(* IEC 61131-3 sources: RegAx/src, 7 files *)

(* ---- RegexCharClass.st ---- *)
NAMESPACE Simatic.Ax.RegAx

    /// Parsed representation of a character class like [abc], [a-z] or [^abc].
    TYPE INTERNAL RegexCharClass : STRUCT
        isNegated : BOOL;
        literalCount : INT;
        literals : ARRAY[1..16] OF CHAR;
        rangeCount : INT;
        ranges : ARRAY[1..8] OF RegexCharClassRange;
    END_STRUCT;
    END_TYPE

END_NAMESPACE

(* ---- RegexCharClassRange.st ---- *)
NAMESPACE Simatic.Ax.RegAx

    /// Inclusive character range used inside a character class.
    TYPE INTERNAL RegexCharClassRange : STRUCT
        rangeStart : CHAR;
        rangeEnd : CHAR;
    END_STRUCT;
    END_TYPE

END_NAMESPACE

(* ---- RegexToken.st ---- *)
NAMESPACE Simatic.Ax.RegAx

    /// Parsed token with optional quantifier information.
    TYPE PUBLIC RegexToken : STRUCT
        tokenType : RegexTokenType;
        literal : CHAR;
        minCount : INT;
        maxCount : INT;
        charClass : RegexCharClass;
    END_STRUCT;
    END_TYPE

END_NAMESPACE

(* ---- RegexTokenType.st ---- *)
NAMESPACE Simatic.Ax.RegAx

    /// Token kinds used by the internal regex tokenizer.
    TYPE PUBLIC RegexTokenType : (
        None,
        Literal,
        DigitClass,
        WordClass,
        CharacterClass,
        EscapedLiteral,
        AnchorStart,
        AnchorEnd
    );
    END_TYPE

END_NAMESPACE

(* ---- Regex.st ---- *)
USING System.Strings;

NAMESPACE Simatic.Ax.RegAx

    /// Public regex facade for configuring a pattern, assigning input and retrieving the match.
    CLASS PUBLIC Regex
        VAR
            /// Pattern used for the next match operation.
            _pattern : STRING;

            /// Input string used for the next match operation.
            _input : STRING;

            /// Last matched substring.
            _match : STRING;

            /// 1-based start index of the last successful match.
            _matchStartIndex : INT;

            /// 1-based end index of the last successful match.
            _matchEndIndex : INT;

            /// Next input position used by MatchNext.
            _nextSearchStartIndex : INT;

            /// Internal tokenizer instance.
            _tokenizer : RegexTokenizer;

            /// Internal matcher instance.
            _matcher : RegexMatcher;
        END_VAR

        /// Stores the regex pattern for subsequent Match calls.
        METHOD PUBLIC SetPattern
            VAR_INPUT
                /// Regex pattern to evaluate.
                pattern : STRING;
            END_VAR
            _pattern := pattern;
        END_METHOD

        /// Stores the input string for subsequent Match calls.
        METHOD PUBLIC SetInput
            VAR_INPUT
                /// Input string to search in.
                inputStr : STRING;
            END_VAR
            _input := inputStr;
            _match := '';
            _matchStartIndex := 0;
            _matchEndIndex := 0;
            _nextSearchStartIndex := 1;
        END_METHOD

        /// Evaluates the configured pattern against the configured input.
        METHOD PUBLIC Match : BOOL
            VAR
                tokens : ARRAY[1..64] OF RegexToken;
                tokenCount : INT;
                anchorStart : BOOL;
                anchorEnd : BOOL;
                inputLength : INT;
                startIndex : INT;
                endIndex : INT;
            END_VAR

            _match := '';
            _matchStartIndex := 0;
            _matchEndIndex := 0;
            _nextSearchStartIndex := 1;
            IF NOT _tokenizer.Tokenize(pattern := _pattern, tokens => tokens, tokenCount => tokenCount, anchorStart => anchorStart, anchorEnd => anchorEnd) THEN
                Match := FALSE;
                RETURN;
            END_IF;

            inputLength := LengthOf(_input);
            IF tokenCount <= 0 THEN
                Match := FALSE;
                RETURN;
            END_IF;

            IF anchorStart THEN
                startIndex := 1;
                IF _matcher.TryMatchFrom(input := _input, startIndex := startIndex, inputLength := inputLength, tokens := tokens, tokenCount := tokenCount, anchorEnd := anchorEnd, endIndex => endIndex) THEN
                    _match := _matcher.BuildMatch(input := _input, startIndex := startIndex, endIndex := endIndex);
                    _matchStartIndex := startIndex;
                    _matchEndIndex := endIndex;
                    _nextSearchStartIndex := endIndex + 1;
                    Match := TRUE;
                    RETURN;
                END_IF;
                Match := FALSE;
                RETURN;
            END_IF;

            startIndex := 1;
            WHILE startIndex <= inputLength DO
                IF _matcher.TryMatchFrom(input := _input, startIndex := startIndex, inputLength := inputLength, tokens := tokens, tokenCount := tokenCount, anchorEnd := anchorEnd, endIndex => endIndex) THEN
                    _match := _matcher.BuildMatch(input := _input, startIndex := startIndex, endIndex := endIndex);
                    _matchStartIndex := startIndex;
                    _matchEndIndex := endIndex;
                    _nextSearchStartIndex := endIndex + 1;
                    Match := TRUE;
                    RETURN;
                END_IF;
                startIndex := startIndex + 1;
            END_WHILE;

            Match := FALSE;
        END_METHOD

        /// Continues searching after the previous successful match.
        METHOD PUBLIC MatchNext : BOOL
            VAR
                tokens : ARRAY[1..64] OF RegexToken;
                tokenCount : INT;
                anchorStart : BOOL;
                anchorEnd : BOOL;
                inputLength : INT;
                startIndex : INT;
                endIndex : INT;
            END_VAR

            _match := '';
            _matchStartIndex := 0;
            _matchEndIndex := 0;

            IF NOT _tokenizer.Tokenize(pattern := _pattern, tokens => tokens, tokenCount => tokenCount, anchorStart => anchorStart, anchorEnd => anchorEnd) THEN
                MatchNext := FALSE;
                RETURN;
            END_IF;

            IF anchorStart OR anchorEnd THEN
                MatchNext := FALSE;
                RETURN;
            END_IF;

            inputLength := LengthOf(_input);
            startIndex := _nextSearchStartIndex;
            IF startIndex < 1 THEN
                startIndex := 1;
            END_IF;

            WHILE startIndex <= inputLength DO
                IF _matcher.TryMatchFrom(input := _input, startIndex := startIndex, inputLength := inputLength, tokens := tokens, tokenCount := tokenCount, anchorEnd := FALSE, endIndex => endIndex) THEN
                    _match := _matcher.BuildMatch(input := _input, startIndex := startIndex, endIndex := endIndex);
                    _matchStartIndex := startIndex;
                    _matchEndIndex := endIndex;
                    _nextSearchStartIndex := endIndex + 1;
                    MatchNext := TRUE;
                    RETURN;
                END_IF;
                startIndex := startIndex + 1;
            END_WHILE;

            MatchNext := FALSE;
        END_METHOD

        /// Returns the substring captured by the last successful Match call.
        METHOD PUBLIC GetMatch : STRING
            GetMatch := _match;
        END_METHOD

        /// Returns the 1-based start index of the last successful match.
        METHOD PUBLIC GetMatchStartIndex : INT
            GetMatchStartIndex := _matchStartIndex;
        END_METHOD

        /// Returns the 1-based end index of the last successful match.
        METHOD PUBLIC GetMatchEndIndex : INT
            GetMatchEndIndex := _matchEndIndex;
        END_METHOD
    END_CLASS

END_NAMESPACE

(* ---- RegexMatcher.st ---- *)
USING System.Strings;

NAMESPACE Simatic.Ax.RegAx

    {axcode:docs-v0:@simatic-ax/regax:Regex.md}
    /// Internal matcher for the supported iterative regex subset.
    CLASS INTERNAL RegexMatcher
        VAR CONSTANT
            /// Maximum length of a returned match.
            MAX_MATCH_LENGTH : INT := 254;
        END_VAR

        /// Tries to match a tokenized pattern against the input string.
        METHOD PUBLIC MatchTokens : BOOL
            VAR_INPUT
                /// Input string to search in.
                input : STRING;

                /// Tokenized regex pattern.
                tokens : ARRAY[1..64] OF RegexToken;

                /// Number of valid tokens.
                tokenCount : INT;

                /// TRUE when matching must start at the beginning of the input.
                anchorStart : BOOL;

                /// TRUE when matching must end at the end of the input.
                anchorEnd : BOOL;
            END_VAR
            VAR_OUTPUT
                /// Matched substring when a match is found.
                matchedText : STRING;
            END_VAR
            VAR
                inputLength : INT;
                startIndex : INT;
                endIndex : INT;
            END_VAR

            MatchTokens := FALSE;
            matchedText := '';
            inputLength := LengthOf(input);

            IF tokenCount <= 0 THEN
                RETURN;
            END_IF;

            IF anchorStart THEN
                startIndex := 1;
                IF THIS.TryMatchFrom(input := input, startIndex := startIndex, inputLength := inputLength, tokens := tokens, tokenCount := tokenCount, anchorEnd := anchorEnd, endIndex => endIndex) THEN
                    matchedText := THIS.BuildMatch(input := input, startIndex := startIndex, endIndex := endIndex);
                    MatchTokens := TRUE;
                END_IF;
                RETURN;
            END_IF;

            startIndex := 1;
            WHILE startIndex <= inputLength DO
                IF THIS.TryMatchFrom(input := input, startIndex := startIndex, inputLength := inputLength, tokens := tokens, tokenCount := tokenCount, anchorEnd := anchorEnd, endIndex => endIndex) THEN
                    matchedText := THIS.BuildMatch(input := input, startIndex := startIndex, endIndex := endIndex);
                    MatchTokens := TRUE;
                    RETURN;
                END_IF;
                startIndex := startIndex + 1;
            END_WHILE;
        END_METHOD

        /// Attempts a match from a specific input position.
        METHOD INTERNAL TryMatchFrom : BOOL
            VAR_INPUT
                /// Input string to search in.
                input : STRING;

                /// 1-based start position for this attempt.
                startIndex : INT;

                /// Cached input length.
                inputLength : INT;

                /// Tokenized regex pattern.
                tokens : ARRAY[1..64] OF RegexToken;

                /// Number of valid tokens.
                tokenCount : INT;

                /// TRUE when the match must consume the full remaining input.
                anchorEnd : BOOL;
            END_VAR
            VAR_OUTPUT
                /// Inclusive end index of the match.
                endIndex : INT;
            END_VAR
            VAR
                tokenIndex : INT;
                inputIndex : INT;
                repeatCount : INT;
                maxAllowed : INT;
            END_VAR

            TryMatchFrom := FALSE;
            endIndex := startIndex - 1;
            inputIndex := startIndex;

            FOR tokenIndex := 1 TO tokenCount DO
                repeatCount := 0;
                maxAllowed := tokens[tokenIndex].maxCount;

                WHILE repeatCount < maxAllowed AND inputIndex <= inputLength DO
                    IF THIS.TokenMatches(token := tokens[tokenIndex], currentChar := input[inputIndex]) THEN
                        repeatCount := repeatCount + 1;
                        inputIndex := inputIndex + 1;
                    ELSE
                        EXIT;
                    END_IF;
                END_WHILE;

                IF repeatCount < tokens[tokenIndex].minCount THEN
                    RETURN;
                END_IF;
            END_FOR;

            endIndex := inputIndex - 1;
            IF anchorEnd AND endIndex <> inputLength THEN
                RETURN;
            END_IF;

            TryMatchFrom := TRUE;
        END_METHOD

        /// Checks whether a single input character satisfies a token.
        METHOD PRIVATE TokenMatches : BOOL
            VAR_INPUT
                /// Token to evaluate.
                token : RegexToken;

                /// Current input character.
                currentChar : CHAR;
            END_VAR
            VAR
                literalIndex : INT;
                rangeIndex : INT;
                isMatch : BOOL;
            END_VAR
            CASE token.tokenType OF
                RegexTokenType#Literal, RegexTokenType#EscapedLiteral:
                    TokenMatches := currentChar = token.literal;
                RegexTokenType#DigitClass:
                    TokenMatches := (currentChar >= '0') AND (currentChar <= '9');
                RegexTokenType#WordClass:
                    TokenMatches := ((currentChar >= 'A') AND (currentChar <= 'Z')) OR ((currentChar >= 'a') AND (currentChar <= 'z')) OR ((currentChar >= '0') AND (currentChar <= '9')) OR (currentChar = '_');
                RegexTokenType#CharacterClass:
                    isMatch := FALSE;
                    FOR literalIndex := 1 TO token.charClass.literalCount DO
                        IF currentChar = token.charClass.literals[literalIndex] THEN
                            isMatch := TRUE;
                            EXIT;
                        END_IF;
                    END_FOR;
                    IF NOT isMatch THEN
                        FOR rangeIndex := 1 TO token.charClass.rangeCount DO
                            IF (currentChar >= token.charClass.ranges[rangeIndex].rangeStart) AND (currentChar <= token.charClass.ranges[rangeIndex].rangeEnd) THEN
                                isMatch := TRUE;
                                EXIT;
                            END_IF;
                        END_FOR;
                    END_IF;
                    IF token.charClass.isNegated THEN
                        TokenMatches := NOT isMatch;
                    ELSE
                        TokenMatches := isMatch;
                    END_IF;
            ELSE
                TokenMatches := FALSE;
            END_CASE;
        END_METHOD

        /// Builds the matched substring from the input indices.
        METHOD INTERNAL BuildMatch : STRING
            VAR_INPUT
                /// Source input string.
                input : STRING;

                /// Inclusive start index of the match.
                startIndex : INT;

                /// Inclusive end index of the match.
                endIndex : INT;
            END_VAR
            VAR
                currentIndex : INT;
                result : STRING;
            END_VAR

            result := '';
            IF endIndex < startIndex THEN
                BuildMatch := result;
                RETURN;
            END_IF;

            FOR currentIndex := startIndex TO endIndex DO
                result := CONCAT(result, input[currentIndex]);
            END_FOR;
            BuildMatch := result;
        END_METHOD
    END_CLASS

END_NAMESPACE

(* ---- RegexTokenizer.st ---- *)
USING System.Strings;

NAMESPACE Simatic.Ax.RegAx

    /// Converts a pattern string into validated regex tokens.
    CLASS INTERNAL RegexTokenizer
        VAR CONSTANT
            /// Maximum number of tokens supported per pattern.
            MAX_TOKEN_COUNT : INT := 64;

            /// Maximum repetition count used for open-ended quantifiers.
            MAX_REPEAT_COUNT : INT := 254;
        END_VAR

        /// Tokenizes the configured regex pattern and extracts anchors.
        METHOD PUBLIC Tokenize : BOOL
            VAR_INPUT
                /// Pattern string to parse.
                pattern : STRING;
            END_VAR
            VAR_OUTPUT
                /// Parsed token sequence.
                tokens : ARRAY[1..64] OF RegexToken;

                /// Number of valid entries in tokens.
                tokenCount : INT;

                /// TRUE when the pattern starts with ^.
                anchorStart : BOOL;

                /// TRUE when the pattern ends with $.
                anchorEnd : BOOL;
            END_VAR
            VAR
                patternLength : INT;
                patternIndex : INT;
                currentChar : CHAR;
                nextChar : CHAR;
                token : RegexToken;
                quantifierStart : INT;
                quantifierEnd : INT;
                repeatMin : INT;
                repeatMax : INT;
                charClassEnd : INT;
            END_VAR

            Tokenize := FALSE;
            tokenCount := 0;
            anchorStart := FALSE;
            anchorEnd := FALSE;
            patternLength := LengthOf(pattern);

            IF patternLength = 0 THEN
                RETURN;
            END_IF;

            patternIndex := 1;
            WHILE patternIndex <= patternLength DO
                currentChar := pattern[patternIndex];

                IF currentChar = '^' THEN
                    IF patternIndex <> 1 THEN
                        RETURN;
                    END_IF;
                    anchorStart := TRUE;
                    patternIndex := patternIndex + 1;
                    CONTINUE;
                END_IF;

                IF currentChar = CHAR#36 THEN
                    IF patternIndex <> patternLength THEN
                        RETURN;
                    END_IF;
                    anchorEnd := TRUE;
                    patternIndex := patternIndex + 1;
                    CONTINUE;
                END_IF;

                token.tokenType := RegexTokenType#None;
                token.literal := CHAR#0;
                token.minCount := 1;
                token.maxCount := 1;
                token.charClass.isNegated := FALSE;
                token.charClass.literalCount := 0;
                token.charClass.rangeCount := 0;

                IF currentChar = CHAR#92 THEN
                    IF patternIndex >= patternLength THEN
                        RETURN;
                    END_IF;

                    patternIndex := patternIndex + 1;
                    nextChar := pattern[patternIndex];
                    CASE nextChar OF
                        'd':
                            token.tokenType := RegexTokenType#DigitClass;
                        'w':
                            token.tokenType := RegexTokenType#WordClass;
                        CHAR#46, CHAR#92, CHAR#94, CHAR#36, CHAR#43, CHAR#63, CHAR#123, CHAR#125, CHAR#40, CHAR#41, CHAR#91, CHAR#93, CHAR#124, CHAR#42:
                            token.tokenType := RegexTokenType#EscapedLiteral;
                            token.literal := nextChar;
                    ELSE
                        RETURN;
                    END_CASE;
                ELSIF currentChar = '[' THEN
                    IF NOT THIS.ParseCharacterClass(pattern := pattern, startIndex := patternIndex, token := token, endIndex => charClassEnd) THEN
                        RETURN;
                    END_IF;
                    patternIndex := charClassEnd;
                ELSIF THIS.IsReserved(currentChar := currentChar) THEN
                    RETURN;
                ELSE
                    token.tokenType := RegexTokenType#Literal;
                    token.literal := currentChar;
                END_IF;

                IF token.tokenType = RegexTokenType#None THEN
                    RETURN;
                END_IF;

                IF tokenCount >= MAX_TOKEN_COUNT THEN
                    RETURN;
                END_IF;

                IF patternIndex < patternLength THEN
                    nextChar := pattern[patternIndex + 1];
                    CASE nextChar OF
                        '?':
                            token.minCount := 0;
                            token.maxCount := 1;
                            patternIndex := patternIndex + 1;
                        '+':
                            token.minCount := 1;
                            token.maxCount := MAX_REPEAT_COUNT;
                            patternIndex := patternIndex + 1;
                        '*':
                            token.minCount := 0;
                            token.maxCount := MAX_REPEAT_COUNT;
                            patternIndex := patternIndex + 1;
                        '{':
                            quantifierStart := patternIndex + 1;
                            IF NOT THIS.ParseQuantifier(pattern := pattern, startIndex := quantifierStart, endIndex => quantifierEnd, repeatMin => repeatMin, repeatMax => repeatMax) THEN
                                RETURN;
                            END_IF;
                            token.minCount := repeatMin;
                            token.maxCount := repeatMax;
                            patternIndex := quantifierEnd;
                    END_CASE;
                END_IF;

                tokenCount := tokenCount + 1;
                tokens[tokenCount] := token;
                patternIndex := patternIndex + 1;
            END_WHILE;

            Tokenize := tokenCount > 0;
        END_METHOD

        /// Returns TRUE for syntax characters that are not accepted as plain literals.
        METHOD PRIVATE IsReserved : BOOL
            VAR_INPUT
                currentChar : CHAR;
            END_VAR
            CASE currentChar OF
                '?', '+', '*', '{', '}', '(', ')', '[', ']', '|':
                    IsReserved := TRUE;
            ELSE
                IsReserved := FALSE;
            END_CASE;
        END_METHOD

        /// Parses a bounded or open-ended repetition quantifier.
        METHOD PRIVATE ParseQuantifier : BOOL
            VAR_INPUT
                /// Full pattern string.
                pattern : STRING;

                /// Index of the opening { character.
                startIndex : INT;
            END_VAR
            VAR_OUTPUT
                /// Index of the closing } character.
                endIndex : INT;

                /// Minimum repetition count.
                repeatMin : INT;

                /// Maximum repetition count.
                repeatMax : INT;
            END_VAR
            VAR
                patternLength : INT;
                currentIndex : INT;
                currentChar : CHAR;
                hasComma : BOOL;
                hasMinDigit : BOOL;
                hasMaxDigit : BOOL;
            END_VAR

            ParseQuantifier := FALSE;
            repeatMin := 0;
            repeatMax := 0;
            endIndex := 0;
            patternLength := LengthOf(pattern);

            IF pattern[startIndex] <> '{' THEN
                RETURN;
            END_IF;

            currentIndex := startIndex + 1;
            WHILE currentIndex <= patternLength DO
                currentChar := pattern[currentIndex];
                IF currentChar >= '0' AND currentChar <= '9' THEN
                    hasMinDigit := TRUE;
                    repeatMin := repeatMin * 10 + (TO_INT(TO_BYTE(currentChar)) - 48);
                    currentIndex := currentIndex + 1;
                ELSE
                    EXIT;
                END_IF;
            END_WHILE;

            IF NOT hasMinDigit THEN
                RETURN;
            END_IF;

            IF currentIndex > patternLength THEN
                RETURN;
            END_IF;

            currentChar := pattern[currentIndex];
            IF currentChar = '}' THEN
                repeatMax := repeatMin;
                endIndex := currentIndex;
                ParseQuantifier := TRUE;
                RETURN;
            END_IF;

            IF currentChar <> ',' THEN
                RETURN;
            END_IF;

            hasComma := TRUE;
            currentIndex := currentIndex + 1;
            WHILE currentIndex <= patternLength DO
                currentChar := pattern[currentIndex];
                IF currentChar >= '0' AND currentChar <= '9' THEN
                    hasMaxDigit := TRUE;
                    repeatMax := repeatMax * 10 + (TO_INT(TO_BYTE(currentChar)) - 48);
                    currentIndex := currentIndex + 1;
                ELSE
                    EXIT;
                END_IF;
            END_WHILE;

            IF currentIndex > patternLength OR pattern[currentIndex] <> '}' THEN
                RETURN;
            END_IF;

            IF hasComma AND NOT hasMaxDigit THEN
                repeatMax := MAX_REPEAT_COUNT;
            END_IF;

            IF repeatMin > repeatMax THEN
                RETURN;
            END_IF;

            endIndex := currentIndex;
            ParseQuantifier := TRUE;
        END_METHOD

        /// Parses a character class expression and stores its literals and ranges.
        METHOD PRIVATE ParseCharacterClass : BOOL
            VAR_INPUT
                /// Full pattern string.
                pattern : STRING;

                /// Index of the opening [ character.
                startIndex : INT;
            END_VAR
            VAR_IN_OUT
                /// Token instance that receives the parsed character class.
                token : RegexToken;
            END_VAR
            VAR_OUTPUT
                /// Index of the closing ] character.
                endIndex : INT;
            END_VAR
            VAR
                patternLength : INT;
                currentIndex : INT;
                currentChar : CHAR;
                nextChar : CHAR;
                hasContent : BOOL;
            END_VAR

            ParseCharacterClass := FALSE;
            endIndex := 0;
            patternLength := LengthOf(pattern);

            IF pattern[startIndex] <> '[' THEN
                RETURN;
            END_IF;

            token.tokenType := RegexTokenType#CharacterClass;
            token.charClass.isNegated := FALSE;
            token.charClass.literalCount := 0;
            token.charClass.rangeCount := 0;

            currentIndex := startIndex + 1;
            IF currentIndex > patternLength THEN
                RETURN;
            END_IF;

            IF pattern[currentIndex] = '^' THEN
                token.charClass.isNegated := TRUE;
                currentIndex := currentIndex + 1;
            END_IF;

            WHILE currentIndex <= patternLength DO
                currentChar := pattern[currentIndex];

                IF currentChar = ']' THEN
                    IF NOT hasContent THEN
                        RETURN;
                    END_IF;
                    endIndex := currentIndex;
                    ParseCharacterClass := TRUE;
                    RETURN;
                END_IF;

                IF currentChar = CHAR#92 THEN
                    RETURN;
                END_IF;

                IF (currentIndex + 2 <= patternLength) AND (pattern[currentIndex + 1] = '-') AND (pattern[currentIndex + 2] <> ']') THEN
                    nextChar := pattern[currentIndex + 2];
                    IF nextChar = CHAR#92 THEN
                        RETURN;
                    END_IF;
                    IF currentChar > nextChar THEN
                        RETURN;
                    END_IF;
                    IF token.charClass.rangeCount >= 8 THEN
                        RETURN;
                    END_IF;
                    token.charClass.rangeCount := token.charClass.rangeCount + 1;
                    token.charClass.ranges[token.charClass.rangeCount].rangeStart := currentChar;
                    token.charClass.ranges[token.charClass.rangeCount].rangeEnd := nextChar;
                    hasContent := TRUE;
                    currentIndex := currentIndex + 3;
                    CONTINUE;
                END_IF;

                IF token.charClass.literalCount >= 16 THEN
                    RETURN;
                END_IF;
                token.charClass.literalCount := token.charClass.literalCount + 1;
                token.charClass.literals[token.charClass.literalCount] := currentChar;
                hasContent := TRUE;
                currentIndex := currentIndex + 1;
            END_WHILE;
        END_METHOD
    END_CLASS

END_NAMESPACE
